(* PLC project v0.6.04_CycleSemiAuto.project, CODESYS CODESYS V3.5 SP19 Patch 1 *)
(* stored: creationDateTime 2026-08-12T05:11:49.748997, modificationDateTime 2026-08-12T05:11:49.748997 *)

(* ═══════════════════════════════════════════════════════════════ 🏗️ ST_HwMachine — Image matérielle brute des entrées communes Machine ─────────────────────────────────────────────────────────────── 📄 Lot L5 (Frontière unique HwIn) 🎨 Regroupe les signaux physiques d'entrée bruts communs à la machine. ═══════════════════════════════════════════════════════════════ *)
TYPE ST_HwMachine : STRUCT
  PowerContactorEngaged_DI : BOOL;  (* Confirm. contacteur puissance engagé *)
  EmergencyChainClosed_DI : BOOL;  (* Boucle AU fermée (coup-de-poing + contact PLC) *)
  PhaseRotationOk_DI : BOOL;  (* Contrôle rotation phases élec. OK *)
  M1_M2_M3_BrakeThermalOk_DI : BOOL;  (* Thermique frein M1/M2/M3 commun OK — 🆕 2026-08-12 : renommé depuis BrakeThermalOk_DI (Device_IO_20260812) *)
  M1_M2_KoboldBottomTouch_DI : BOOL;  (* Retour détecteur fond Kobold — 🆕 2026-08-12 : renommé depuis M1_M2_KoboldContactFond_DI (Device_IO_20260812) *)
  HydraulicThermalOk_DI : BOOL;  (* Thermique centrale hydraulique OK *)
  ConveyorInfeedReady_DI : BOOL;  (* Autorisation démarrage crible (dépôt gravats) *)
  HopperFull_OR_GateRaised_DI : BOOL;  (* 🆕 2026-08-12 : Trémie pleine OU grille levée — pas encore câblé électriquement, *)
END_STRUCT;
END_TYPE
